FUNCTION_BLOCK CommonDedicatedSel (* Basic Function Block Type *)
  (* Standard: 61499-2 *)
  (* Version 0.0, 8/19/2026, Schneider Electric, Template *)
  PACKAGE SE.Nereda;
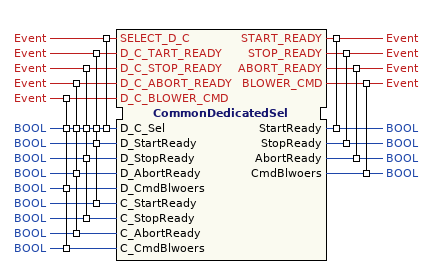
  EVENT_INPUT
    SELECT_D_C WITH D_C_Sel;
    D_C_TART_READY WITH D_StartReady, D_C_Sel, C_StartReady; (* Normal Execution Request *)
    D_C_STOP_READY WITH D_StopReady, D_C_Sel, C_StopReady;
    D_C_ABORT_READY WITH D_AbortReady, D_C_Sel, C_AbortReady;
    D_C_BLOWER_CMD WITH D_CmdBlwoers, D_C_Sel, C_CmdBlwoers;
  END_EVENT
  EVENT_OUTPUT
    START_READY WITH StartReady;
    STOP_READY WITH StopReady;
    ABORT_READY WITH AbortReady;
    BLOWER_CMD WITH CmdBlwoers;
  END_EVENT
  VAR_INPUT
    D_C_Sel : BOOL; (* FALSE = Dedicated | TRUE = Common *)
    D_StartReady : BOOL;
    D_StopReady : BOOL;
    D_AbortReady : BOOL;
    D_CmdBlwoers : BOOL;
    C_StartReady : BOOL;
    C_StopReady : BOOL;
    C_AbortReady : BOOL;
    C_CmdBlwoers : BOOL;
  END_VAR
  VAR_OUTPUT
    StartReady : BOOL;
    StopReady : BOOL;
    AbortReady : BOOL;
    CmdBlwoers : BOOL;
  END_VAR
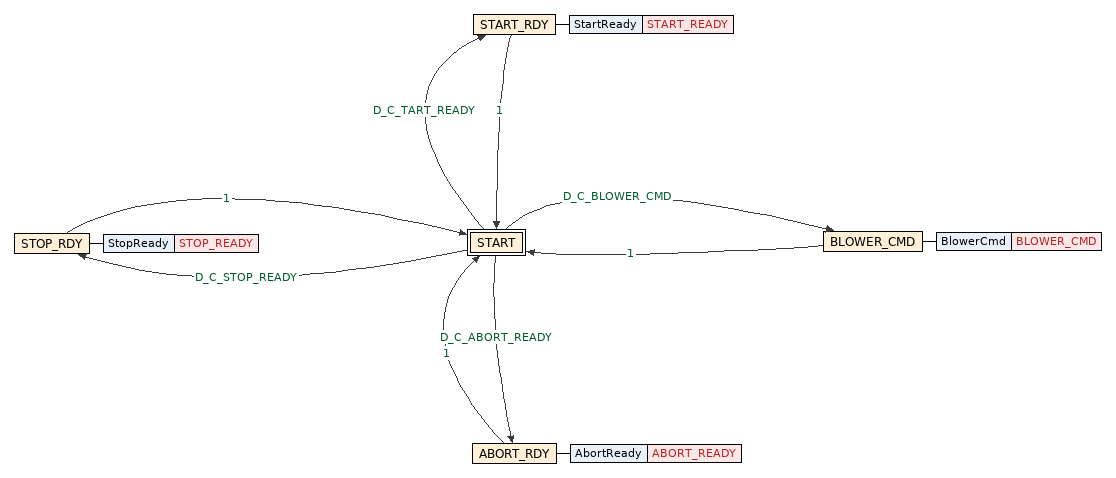
  EC_STATES
    START; (* Initial State *)
    START_RDY : StartReady -> START_READY;
    STOP_RDY : StopReady -> STOP_READY;
    ABORT_RDY : AbortReady -> ABORT_READY;
    BLOWER_CMD : BlowerCmd -> BLOWER_CMD;
  END_STATES
  EC_TRANSITIONS
    START TO START_RDY := D_C_TART_READY;
    START_RDY TO START := 1;
    START TO STOP_RDY := D_C_STOP_READY;
    STOP_RDY TO START := 1;
    START TO ABORT_RDY := D_C_ABORT_READY;
    ABORT_RDY TO START := 1;
    START TO BLOWER_CMD := D_C_BLOWER_CMD;
    BLOWER_CMD TO START := 1;
  END_TRANSITIONS
  ALGORITHM StartReady IN ST:
;
IF D_C_Sel THEN
	StartReady := C_StartReady;
ELSE
	StartReady := D_StartReady;
END_IF;
  END_ALGORITHM
  ALGORITHM StopReady IN ST:
;
IF D_C_Sel THEN
	StopReady := C_StopReady;
ELSE
	StopReady := D_StopReady;
END_IF;
  END_ALGORITHM
  ALGORITHM BlowerCmd IN ST:
;
IF D_C_Sel THEN
	CmdBlwoers := C_CmdBlwoers;
ELSE
	CmdBlwoers := D_CmdBlwoers;
END_IF;
  END_ALGORITHM
  ALGORITHM AbortReady IN ST:
;
IF D_C_Sel THEN
	AbortReady := C_AbortReady;
ELSE
	AbortReady := D_AbortReady;
END_IF;
  END_ALGORITHM
END_FUNCTION_BLOCK
